FUNCTION_BLOCK TEST_CONDITION (* Service Interface Function Block Type *)
  (* Standard: 61499-2; Description: Copyright (c) 2019 fortiss GmbH This program and the accompanying materials are made available under the terms of the Eclipse Public License 2.0 which is available at https://www.eclipse.org/legal/epl-2.0/ SPDX-License-Identifier: PL-2.0 *)
  (* Version 3.0, 2025-04-14, Patrick Aigner, changed package *)
  (* Version 1.0, 2019-01-16, Jose Cabral, fortiss GmbH *)
  PACKAGE eclipse4diac::utils;
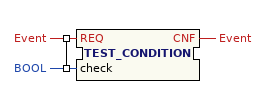
  EVENT_INPUT
    REQ WITH check; (* Request Test *)
  END_EVENT
  EVENT_OUTPUT
    CNF; (* Test finished *)
  END_EVENT
  VAR_INPUT
    check : BOOL; (* Test fails if check == 0, passes otherwise *)
  END_VAR
END_FUNCTION_BLOCK
